FUNCTION_BLOCK FB_SOLVEABCDE
VAR_INPUT
	alfa : REAL:= 0; //ángulo del brazo pxosimal izquierdo
	beta : REAL:= 0; //ángulo del brazo pxosimal derecho
END_VAR
VAR_OUTPUT
	
	Xa : REAL:= 0; 
	Ya : REAL:= 0; 
	Xb : REAL:= 0; 
	Yb : REAL:= 0; 
	Xc : REAL:= 0; 
	Yc : REAL:= 0;
	Xd : REAL:= 0; 
	Yd : REAL:= 0; 
	Xe : REAL:= 0; 
	Ye : REAL:= 0; 
	error : BOOL :=0;
	check_AB : REAL:=GVL.l1;
	check_BC : REAL:=GVL.l2;
	check_CD : REAL:=GVL.l2;
	check_DE : REAL:=GVL.l1;
	

END_VAR
VAR
	aux1 : REAL;
	aux2 : REAL;
	A : REAL;
	B : REAL;
	C : REAL;
END_VAR

error:=FALSE;

// A
Xa := -GVL.d ;
Ya := 0 ;

//B
Xb := Xa + GVL.l1*COS(alfa);
Yb := GVL.l1*SIN(alfa);

//E
Xe := GVL.d ;
Ye := 0 ;

//D
Xd := Xe + GVL.l1*COS(beta);
Yd := GVL.l1*SIN(beta);

//Chekcs
IF SQRT((Xd-Xb)*(Xd-Xb)+(Yd-Yb)*(Yd-Yb))>2*GVL.l2 THEN //B y D demaisado separados
	error:=TRUE;
	ELSE IF Xb>=Xd THEN //brazos proximales cruzados
		error:=TRUE;
		ELSE //calculate Xc
			aux1:=(Xb*Xb-Xd*Xd+Yb*Yb-Yd*Yd)/(2*(Xb-Xd));
			aux2:=-(Yb-Yd)/(Xb-Xd);
			A:=1+ aux2*aux2 ;
			B:=2*(aux1*aux2-Xb*aux2-Yb);
			C:=aux1*aux1-2*Xb*aux1+Yb*Yb+Xb*Xb-GVL.l2*GVL.l2;
			Yc := (-B+SQRT(B*B-4*A*C))/(2*A);
			Xc := aux1+aux2*Yc;
		END_IF
		
check_AB:=SQRT((Xb-Xa)*(Xb-Xa)+(Yb-Ya)*(Yb-Ya));
check_BC:=SQRT((Xb-Xc)*(Xb-Xc)+(Yb-Yc)*(Yb-Yc));
check_CD:=SQRT((Xd-Xc)*(Xd-Xc)+(Yd-Yc)*(Yd-Yc));
check_DE:=SQRT((Xd-Xe)*(Xd-Xe)+(Yd-Ye)*(Yd-Ye));
		
	END_IF

END_FUNCTION_BLOCK

(* stored: Version 1.1.0.1, ProductVersion 3.1.4024.4
   POU FB_SOLVEABCDE: Id {1478d989-93c2-4a9b-9880-0970096e4db9}, SpecialFunc None *)
